TYPE DUT_UpdateCuttersOnDrum :
STRUCT
	Drum		: STRING(30);
	JsonValue	: STRING(DB.MAX_STRING_SIZE);
END_STRUCT
END_TYPE

(* stored: Version 1.1.0.1, ProductVersion 3.1.4024.15
   DUT DUT_UpdateCuttersOnDrum: Id {955717c0-7145-4102-a2ca-ecbfbaca4823} *)
